PROGRAM PRG_2_PMPS
VAR
    fbArbiterIO: FB_SubSysToArbiter_IO;
END_VAR


GVL_PMPS.fbFastFaultOutput1.Execute();
GVL_PMPS.fbFastFaultOutput2.Execute();
fbArbiterIO(
    Arbiter:=GVL_PMPS.fbArbiter,
    fbFFHWO:=GVL_PMPS.fbFastFaultOutput1);

END_PROGRAM

(* stored: Version 1.1.0.1, ProductVersion 3.1.4022.18
   POU PRG_2_PMPS: Id {b84dea55-5b52-40eb-8f1a-0d90375bdbc2}, SpecialFunc None *)
